// TIA Portal V19 export
VAR_GLOBAL   // PLC tag table "Default tag table_3"
   A0302_Rulliera_Lato_1_Testa_Phc_PezzoCentraturaCentrale AT %I311.1 : Bool;   // 2010BF1
END_VAR
